(*
Nazwa:		FB_WeightStation
Opis:		Podnoszenie wag
Wersja:		V0.26
Data:		04.09.2024
Autor:		DP, 
Urządzenia:	Siłowniki
Ostatnie zmiany:
	- 20250904 [DP] EventLog-do sprawdzenia, 1 spr->wywołać błędy 
	- 2024-10-01 [DP] Liczniki po Aborting
	- 2024-04-17 [DP] Przerobienie liczenia i uprowszenie, dwufaz

Konfiguracja:
	- Krokówka
	Instukcja:
		-
		-
	
Info:
	- 
*)

FUNCTION_BLOCK FB_WeightStation
VAR_INPUT
	bEnable											: BOOL;
	bEStop											: BOOL;
	bRun											: BOOL;

	bTwoPhaseMode									: BOOL;
	bCountingBeforeSensorsMode						: BOOL;
    eGlobalState        							: E_PMLState; 							//Stan ogólny maszyny, tylko do błędu
	bConveyorRunning								: BOOL;									//Transporter pracuje, tylko do błędu
	bWeight1ActuatorSensorUp						: BOOL;									//Pierwsza waga podniesiona
	bWeight1FormSensor								: BOOL;									//Obecność formatki na pierwszej wadze     
	bWeight1FormBeforeSensor						: BOOL;									//Obecność formatki przed pierwszą wagą 

	bWeight2ActuatorSensorUp						: BOOL;									//Druga waga podniesiona
	bWeight2FormSensor								: BOOL;									//Obecność formatki na drugiek wadze
	bWeight2FormBeforeSensor						: BOOL;									//Obecność formatki przed pierwszą wagą 
	
	bWeight3ActuatorSensorUp						: BOOL;									//Trzecia waga podniesiona
	bWeight3FormSensor								: BOOL;									//Obecność formatki na trzeciej wadze
	bWeight3FormBeforeSensor						: BOOL;									//Obecność formatki przed pierwszą wagą 
	
	bWeight4ActuatorSensorUp						: BOOL;									//Czwarta waga podniesiona
	bWeight4FormSensor								: BOOL;									//Obecność formatki na czwartej wadze
	bWeight4FormBeforeSensor						: BOOL;									//Obecność formatki przed pierwszą wagą 
	
	bCanReleaseForms								: BOOL;									//Można wypuścić formatki
	bWeighingCycle									: BOOL;									//Trwa ważenie
                                    	
	arrWeightPackageState							: ARRAY [1..17] OF S_PackageState;		//Rejestr nad wagami
	
	bResetCycle										: BOOL;									//Reset cyklu
	
	bHoming											: BOOL;
	bIgnoreError									: BOOL;
	bReset											: BOOL;
	bManualMovement									: BOOL;
	                                    			
	_TIMERS_										: BOOL;
	tWeight1ActuatorUpDelay							: TIME;									//Opóźnienie podnoszenia wagi 1
	tWeight2ActuatorUpDelay							: TIME;									//Opóźnienie podnoszenia wagi 2
	tWeight3ActuatorUpDelay							: TIME;									//Opóźnienie podnoszenia wagi 3
	tWeight4ActuatorUpDelay							: TIME;									//Opóźnienie podnoszenia wagi 4
	
	_ALARMINFO_										: BOOL;
	udiStationIndex									: UDINT;								//Numer stacji
	sStationName									: WSTRING;
	
END_VAR   
                              			
VAR_OUTPUT                              			
	eState											: E_Station;							//Stan ogólny bloku
	eRunningState									: E_WeightLiftStationState;				//Stan stacji
	
	bWeight1Actuator								: BOOL;									//Podnoszenie 1 wagi
	bWeight2Actuator								: BOOL;									//Podnoszenie 2 wagi
	bWeight3Actuator								: BOOL;									//Podnoszenie 3 wagi
	bWeight4Actuator								: BOOL;									//Podnoszenie 4 wagi

	iFormsCounterWeight1							: INT;									//Licznik formatek
	iFormsCounterWeight2							: INT;									//Licznik formatek na wadze 2
	iFormsCounterWeight3							: INT;									//Licznik formatek na wadze 3
	iFormsCounterWeight4							: INT;									//Licznik formatek na wadze 4
	
	bError											: BOOL;									//Błąd stacji
	udiErrorID										: UDINT;								//Numer błędu
	sErrorDescription								: STRING(255);							//Opis błędu
	sErrorDescription2								: STRING(200);							//Opis błędu
	sErrorStationName								: STRING(200);							//Nazwa stacji
	udiStationID									: UDINT;								// Nr stacji
                                    			
	tCycleTime										: TIME;									//Czas cyklu
	bHomingDone										: BOOL;									//Stacja zbazowana 
	bWeighingCycleDone								: BOOL;									//Koniec ważenia 
	bCycleDone										: BOOL;									//Cykl skończony 			
	bTareWeights									: BOOL;		
END_VAR

VAR_IN_OUT
	bManualWeight1Actuator							: BOOL;									//Tryb manualny, Waga 1 UP	
	bManualWeight2Actuator							: BOOL;									//Tryb manualny, Waga 2 UP
	bManualWeight3Actuator							: BOOL;									//Tryb manualny, Waga 3 UP
	bManualWeight4Actuator							: BOOL;									//Tryb manualny, Waga 4 UP	
	bDeparture										: BOOL;					
	bAutoTare										: BOOL;	
END_VAR

VAR
	eLastStateTemp									: E_Station;							//Ostatni stan CONTROL
	eLastState										: E_Station;							//Ostatni stan CONTROL
	eLastRunningStateTemp							: E_WeightLiftStationState;				//Ostatni stan Running
	eLastRunningState								: E_WeightLiftStationState;				//Ostatni stan Running
	eRunningStateBeforeEStop	             		: E_WeightLiftStationState;	                      			                                    		
	tonWeight1ActuatorDelay							: TON;									//TON, opóźnienie podnoszenia wagi 1
	tonWeight2ActuatorDelay							: TON;									//TON, opóźnienie podnoszenia wagi 2
	tonWeight3ActuatorDelay							: TON;									//TON, opóźnienie podnoszenia wagi 3
	tonWeight4ActuatorDelay							: TON;									//TON, opóźnienie podnoszenia wagi 4
	tonWeightAntuatorOffDelay						: TON;
	tonPreparingToReadyDelay						: TON;
	tonResetting									: TON;
	tofRunning										: TOF;
	rtResetCommands									: R_TRIG;
	tonHoming 										: TON;
	tonReadyAndRepair								: TON;					
	tonAbortedDelay									: TON;
	tonRepairDelay									: TON;									//TON, czas po którym przechodzimy do naprawy
	tonRepairOnDelay								: TON;									//TON, czas na wyjazd wszystkich formatek
	rtWeight1FormSensor								: R_TRIG;								//R_Trig, zbocze nar (przy wadze 1)
	rtWeight2FormSensor								: R_TRIG;								//R_Trig, zbocze nar (przy wadze 2)
	rtWeight3FormSensor								: R_TRIG;								//R_Trig, zbocze nar (przy wadze 3)
	rtWeight4FormSensor								: R_TRIG;								//R_Trig, zbocze nar (przy wadze 4)

	ftWeight1FormBeforeSensor						: F_TRIG;								
	ftWeight2FormBeforeSensor						: F_TRIG;								
	ftWeight3FormBeforeSensor						: F_TRIG;								
	ftWeight4FormBeforeSensor						: F_TRIG;								
	
	tonWeightsEmpty									: TON;
	toniCaseTareWeights1							: TON;
	toniCaseTareWeights2							: TON;
	
	bLastStateWeight1Actuator						: BOOL;							
	bLastStateWeight2Actuator						: BOOL;	
	bLastStateWeight3Actuator						: BOOL;	
	bLastStateWeight4Actuator						: BOOL;	
	
	bStateError										: BOOL;
	bWasAborting									: BOOL;
	
	bRepairAllRegistersAreEmpty						: BOOL;								
	
	//Błedy
	bResetCycleOn									: BOOL;
	tonWeight1ActuatorUpError 						: TON;
	tonWeight2ActuatorUpError 						: TON;
	tonWeight3ActuatorUpError 						: TON;
	tonWeight4ActuatorUpError 						: TON;
	
	//Śmiecie
	tonRepair1: TON;
	tonRepair2: TON;
	tonRepair3: TON;
	tonRepair4: TON;
	tonRepair5: TON;
	tonRepair6: TON;
	
	rtrigCycleTimerRead: R_TRIG;
	tonCycleTimer: TON;
	tt: INT;
	rtWeight3FormSensorWithDelay2: R_TRIG;

	iRepair1: INT;
	iRepair2: INT;
	iRepair3: INT;
	iRepair4: INT;
	iRepair5: INT;
	iRepair6: INT;
	
	tofRunningStopping: TOF;
	iCaseTareWeights:INT;
	
	//Zmienne od EVENTLOGGER
	bAlarmInit 						: BOOL := TRUE; 
	nAlarmNumerator					: INT;
	arfbAlarm						: ARRAY[0..19] OF  FB_TcAlarm;		//Tablica bloczków błędów
	fbSourceInfo 					: FB_TcSourceInfo;
	iSourceInfo						: I_TcSourceInfo;
	sAlarmTest						: STRING;
	tonEventLogger					: TON;
	//Koniec zmiennych od EVENTLOGGER
	bTest							: BOOL;
END_VAR

ResetAll();
ACT_ErrorHandling();
ACT_Signals();
aRepair();
ACT_Control();
ACT_Statistics();
aStationID();

IF eLastStateTemp <> eState THEN
	eLastState							:= eLastStateTemp;
END_IF
eLastStateTemp							:= eState;

IF eLastRunningStateTemp <> eRunningState THEN
	eLastRunningState					:= eLastRunningStateTemp;
END_IF
eLastRunningStateTemp					:= eRunningState;

ACTION ACT_Control:


	(*****Wyłączenie enable*****)
	IF NOT bEnable AND NOT bError THEN
		IF eState <> E_Station.eDisabled AND eState <> E_Station.ePreparingToDisable THEN
				eState 								:= E_Station.ePreparingToDisable; 
		END_IF	
	END_IF

	(*****Estop*****)
	IF NOT bEstop  THEN	
		IF eState <> E_Station.eAborted AND eState <> E_Station.eAborting AND eState <> E_Station.eDisabled THEN
				eRunningStateBeforeEStop			:= eRunningState;
				eState 								:= E_Station.eAborting; 
		END_IF
	END_IF


CASE eState OF
	
	
	E_Station.eDisabled: 					// Stan nieaktywnosci (Stacja wyłączona)
		IF bEnable THEN
			eState											:= E_Station.ePreparingToReady;
		END_IF	
	//------------------------------------------------------------------------------
	
	E_Station.eAborted: 					// Stan bezpiecznego zatrzymania (po Abortingu)			
		IF bEStop THEN
			eState											:= E_Station.ePreparingToReady;
		END_IF	
	//------------------------------------------------------------------------------
	
	E_Station.eAborting:                 	// Stan bezpiecznego zatrzymywania (po EStopie)
	
		aResetCommandsAborting();
		bWasAborting										:= TRUE;
		eState												:= E_Station.eAborted;	
		eRunningState										:= E_WeightLiftStationState.eReady;
	//------------------------------------------------------------------------------
	
	E_Station.eError:                 	 	// Stan błędu 	
	
		IF bReset THEN
			eState									:= E_Station.eResetting;	
		ELSE
			aResetCommands();
		END_IF
		
	//------------------------------------------------------------------------------

	
	E_Station.eResetting:					// Stan resetowania bledu (po Errorze)

// 		CASE udiErrorID OF 
// //		CASE udiErrorID - udiStationIndex OF 
// 			
// 			191,195: //Error 1
// 				bWeight1Actuator						:=	FALSE;
// 				bError									:=	FALSE;
// 			192,196://Error 2
// 				bWeight2Actuator						:=	FALSE;
// 				bError									:=	FALSE;	
// 			193: //Error 3
// 				bWeight3Actuator						:=	FALSE;
// 				bError									:=	FALSE;
// 			194: //Error 4
// 				bWeight4Actuator						:=	FALSE;
// 				bError									:=	FALSE;			
// 			
// 		END_CASE

		bWeight1Actuator						:=	FALSE;
		bWeight2Actuator						:=	FALSE;		
		bWeight3Actuator						:=	FALSE;
		bWeight4Actuator						:=	FALSE;		

		IF NOT bError THEN
			udiErrorID										:= 0;
			sErrorDescription								:= '';
			sErrorDescription2								:= '';
			eState											:= E_Station.ePreparingToReady;
		ELSIF tonResetting.Q THEN                   	
			eState											:= E_Station.eError;
		END_IF
	//------------------------------------------------------------------------------
	E_Station.eManualMovement:     			// Stan ruchów manualnych  
	
		ACT_ManualMovements();
		//Wyjście z trybu serwisowego
		IF NOT bManualMovement THEN
			bWeight1Actuator								:=	bLastStateWeight1Actuator;
			bWeight2Actuator								:=	bLastStateWeight2Actuator;
			bWeight3Actuator								:=	bLastStateWeight3Actuator;
			bWeight4Actuator								:=	bLastStateWeight4Actuator;
			eState											:=	E_Station.eReady;
		END_IF
	//------------------------------------------------------------------------------
	
	E_Station.eHoming:						// Stan bazowania
	
		ACT_Homing();
		IF NOT bHoming AND tonHoming.Q THEN
			eState									:=	E_Station.ePreparingToReady;
		END_IF	
	//------------------------------------------------------------------------------
	
	E_Station.eHomingDone:                  // Stan wykonania bazowania
	
		bHomingDone											:= TRUE;		
		IF NOT bHoming THEN
			eState											:= E_Station.eReady;
		END_IF	
	//------------------------------------------------------------------------------
	
	
	E_Station.ePreparingToReady:            // Stan przygotowywania do gotowosci (zawsze przed Ready)
		//bHomingDone										:=	FALSE;	
		bWeight1Actuator									:=	FALSE;
		bWeight2Actuator									:=	FALSE;
		bWeight3Actuator									:=	FALSE;
		bWeight4Actuator									:=	FALSE;
		
		IF NOT bWasAborting THEN
			iFormsCounterWeight1								:= 3;	
			iFormsCounterWeight2								:= 2;
			iFormsCounterWeight3								:= 1;
			iFormsCounterWeight4								:= 0;
		END_IF
		
		IF tonPreparingToReadyDelay.Q THEN
			eState											:= E_Station.eReady;
		END_IF	
		
	//------------------------------------------------------------------------------
	
	
	E_Station.ePreparingToDisable:          // Stan przygotowywania do nieaktywnosci (po wyłączeniu Enable)	
		
		bWeight1Actuator									:=	FALSE;
		bWeight2Actuator									:=	FALSE;
		bWeight3Actuator									:=	FALSE;
		bWeight4Actuator									:=	FALSE;
		
		iFormsCounterWeight1								:= 3;	
		iFormsCounterWeight2								:= 2;
		iFormsCounterWeight3								:= 1;
		iFormsCounterWeight4								:= 0;
					
		eState												:= E_Station.eDisabled;
		eRunningState										:= E_WeightLiftStationState.eDisabled;
		
	//------------------------------------------------------------------------------
	
	
	E_Station.eReady:						// Stan gotowosci
		bWasAborting										:= FALSE;
		IF (bRun OR bAutoTare) AND bHomingDone AND NOT bCycleDone THEN
			eRunningState									:= E_WeightLiftStationState.eReady;
			eState											:= E_Station.eStarting;
		END_IF
		
		IF bHoming THEN
			eState											:= E_Station.eHoming;
		END_IF
		
		IF bManualMovement THEN
			bLastStateWeight1Actuator	:=	bManualWeight1Actuator	:=	bWeight1Actuator;
			bLastStateWeight2Actuator	:=	bManualWeight2Actuator	:=	bWeight2Actuator;
			bLastStateWeight3Actuator	:=	bManualWeight3Actuator	:=	bWeight3Actuator;
			bLastStateWeight4Actuator	:=	bManualWeight4Actuator	:=	bWeight4Actuator;		
			eState											:= E_Station.eManualMovement;
		END_IF
		
		IF NOT bRun THEN
			bCycleDone										:= FALSE;
		END_IF
		IF tonReadyAndRepair.Q THEN
			eRunningState									:= E_WeightLiftStationState.eReady;
		END_IF
	//------------------------------------------------------------------------------
	
	
	E_Station.eStopping:					// Stan zatrzymywania 

		ACT_Running();
		eState											:= E_Station.eReady;
		eRunningState									:= E_WeightLiftStationState.eReady;
		
		
	//------------------------------------------------------------------------------
	
	
	E_Station.eStarting:                  	// Stan uruchamiania (po Ready)
	
		eState												:= E_Station.eRunning;
	//------------------------------------------------------------------------------
	
	
	E_Station.eRunning:               		// Stan wykonywania cyklu (po Startingu), w tym stanie osobny
		
		ACT_Running();
		
		IF NOT bRun THEN
			eState											:= E_Station.eStopping;
		END_IF
		
		IF bCycleDone THEN
			eState											:= E_Station.eReady;
		END_IF
	//------------------------------------------------------------------------------
	
	
END_CASE
END_ACTION

ACTION ACT_ErrorHandling:
// Alarm_0300	300	Error	Podnoszenie wagi nr 1 | Blokada podnoszenia siłownika - sprawdź czujnik lub odblokuj
// Alarm_0301	301	Error	Podnoszenie wagi nr 2 | Blokada podnoszenia siłownika - sprawdź czujnik lub odblokuj
// Alarm_0302	302	Error	Podnoszenie wagi nr 3 | Blokada podnoszenia siłownika - sprawdź czujnik lub odblokuj
// Alarm_0303	303	Error	Podnoszenie wagi nr 4 | Blokada podnoszenia siłownika - sprawdź czujnik lub odblokuj
// Alarm_0304	304	Error	Podnoszenie wagi nr 5 | Blokada podnoszenia siłownika - sprawdź czujnik lub odblokuj
// Alarm_0305	305	Error	Podnoszenie wagi nr 6 | Blokada podnoszenia siłownika - sprawdź czujnik lub odblokuj

IF bAlarmInit THEN
    bAlarmInit := FALSE; 
	fbSourceInfo.Clear();
	fbSourceInfo.sName:=wsLiteral_TO_UTF8(sStationName);//'Machine';
	fbSourceInfo.nId:=udiStationIndex;//2700;
	// Alarm_0300	300	Error	Podnoszenie wagi nr 1 | Blokada podnoszenia siłownika - sprawdź czujnik lub odblokuj
    arfbAlarm[0].CreateEx(stEventEntry := TC_EVENTS.AlarmClass.Alarm_0300, bWithConfirmation:= FALSE,  ipSourceInfo:= fbSourceInfo); 
	// Alarm_0301	301	Error	Podnoszenie wagi nr 2 | Blokada podnoszenia siłownika - sprawdź czujnik lub odblokuj
	arfbAlarm[1].CreateEx(stEventEntry := TC_EVENTS.AlarmClass.Alarm_0301, bWithConfirmation:= FALSE,  ipSourceInfo:= fbSourceInfo);
	// Alarm_0302	302	Error	Podnoszenie wagi nr 3 | Blokada podnoszenia siłownika - sprawdź czujnik lub odblokuj
	arfbAlarm[2].CreateEx(stEventEntry := TC_EVENTS.AlarmClass.Alarm_0302, bWithConfirmation:= FALSE,  ipSourceInfo:= fbSourceInfo);
	// Alarm_0303	303	Error	Podnoszenie wagi nr 4 | Blokada podnoszenia siłownika - sprawdź czujnik lub odblokuj
	arfbAlarm[3].CreateEx(stEventEntry := TC_EVENTS.AlarmClass.Alarm_0303, bWithConfirmation:= FALSE,  ipSourceInfo:= fbSourceInfo);
	// Alarm_0304	304	Error	Podnoszenie wagi nr 5 | Blokada podnoszenia siłownika - sprawdź czujnik lub odblokuj
	arfbAlarm[4].CreateEx(stEventEntry := TC_EVENTS.AlarmClass.Alarm_0304, bWithConfirmation:= FALSE,  ipSourceInfo:= fbSourceInfo);
	// Alarm_0305	305	Error	Podnoszenie wagi nr 6 | Blokada podnoszenia siłownika - sprawdź czujnik lub odblokuj
	arfbAlarm[5].CreateEx(stEventEntry := TC_EVENTS.AlarmClass.Alarm_0305, bWithConfirmation:= FALSE,  ipSourceInfo:= fbSourceInfo);
END_IF

bStateError								:= (eState = E_Station.eError) OR (eState = E_Station.eResetting);

tonEventLogger (IN:= NOT tonEventLogger.Q, PT:=T#1S);

IF tonEventLogger.Q THEN
	
	// Alarm_0300	300	Error	Podnoszenie wagi nr 1 | Blokada podnoszenia siłownika - sprawdź czujnik lub odblokuj
	// Alarm_0304	304	Error	Podnoszenie wagi nr 5 | Blokada podnoszenia siłownika - sprawdź czujnik lub odblokuj
	//Błąd podnoszenia wagi 1 
	tonWeight1ActuatorUpError				(IN:= bWeight1Actuator AND NOT bWeight1ActuatorSensorUp	, PT:=T#2S);
	IF tonWeight1ActuatorUpError.Q THEN
		IF NOT bTwoPhaseMode AND NOT arfbAlarm[0].bActive THEN
			arfbAlarm[0].Raise(nTimeStamp:=0);
		END_IF
		IF bTwoPhaseMode AND NOT arfbAlarm[4].bActive THEN
				arfbAlarm[4].Raise(nTimeStamp:=0);
		END_IF
		IF (arfbAlarm[0].bActive OR arfbAlarm[4].bActive) AND bReset THEN
			bWeight1Actuator			:= FALSE;
		END_IF
		ELSE	
		IF NOT bTwoPhaseMode AND arfbAlarm[0].bActive AND bReset THEN
			arfbAlarm[0].Clear(nTimeStamp:=0, bResetConfirmation:= FALSE);
		END_IF
		IF bTwoPhaseMode AND arfbAlarm[4].bActive AND bReset THEN
			arfbAlarm[4].Clear(nTimeStamp:=0, bResetConfirmation:= FALSE);
		END_IF
	// 	bError								:= TRUE;
	// 	IF NOT bTwoPhaseMode THEN
	// 	udiErrorID							:= 191;	
	// 	//udiErrorID 						:= udiErrorID + udiStationIndex;
	// 	sErrorDescription					:= 'Podnoszenie wagi nr 1';
	// 	END_IF
	// 	
	// 	IF bTwoPhaseMode THEN
	// 		udiErrorID						:= 195;
	// 		sErrorDescription				:= 'Podnoszenie wagi nr 5';
	// 	END_IF
	// 	sErrorDescription2					:= 'Blokada podnoszenia siłownika - sprawdź czujnik lub odblokuj';
	END_IF
	// Alarm_0301	301	Error	Podnoszenie wagi nr 2 | Blokada podnoszenia siłownika - sprawdź czujnik lub odblokuj
	// Alarm_0305	305	Error	Podnoszenie wagi nr 6 | Blokada podnoszenia siłownika - sprawdź czujnik lub odblokuj
	//Błąd podnoszenia wagi 2
	tonWeight2ActuatorUpError				(IN:= bWeight2Actuator AND NOT bWeight2ActuatorSensorUp	, PT:=T#2S);
	IF tonWeight2ActuatorUpError.Q THEN
		
		IF NOT bTwoPhaseMode AND NOT arfbAlarm[1].bActive THEN
				arfbAlarm[1].Raise(nTimeStamp:=0);
		END_IF
		IF bTwoPhaseMode AND NOT arfbAlarm[5].bActive THEN
				arfbAlarm[5].Raise(nTimeStamp:=0);
		END_IF	
		IF (arfbAlarm[1].bActive OR arfbAlarm[5].bActive) AND bReset THEN
			bWeight1Actuator			:= FALSE;
		END_IF
		ELSE	
		IF NOT bTwoPhaseMode AND arfbAlarm[1].bActive AND bReset THEN
			arfbAlarm[1].Clear(nTimeStamp:=0, bResetConfirmation:= FALSE);
		END_IF	
		IF bTwoPhaseMode AND arfbAlarm[5].bActive AND bReset THEN
			arfbAlarm[5].Clear(nTimeStamp:=0, bResetConfirmation:= FALSE);
		END_IF	
	// 	bError								:= TRUE;
	// 	IF NOT bTwoPhaseMode THEN
	// 	udiErrorID							:= 192;	
	// 	//udiErrorID 						:= udiErrorID + udiStationIndex;
	// 	sErrorDescription					:= 'Podnoszenie wagi nr 2';
	// 	END_IF
	
	// 	IF bTwoPhaseMode THEN
	// 		udiErrorID						:= 196;
	// 		sErrorDescription				:= 'Podnoszenie wagi nr 6';
	// 	END_IF
	// 	sErrorDescription2					:= 'Blokada podnoszenia siłownika - sprawdź czujnik lub odblokuj';	
	END_IF
	// Alarm_0302	302	Error	Podnoszenie wagi nr 3 | Blokada podnoszenia siłownika - sprawdź czujnik lub odblokuj
	//Błąd podnoszenia wagi 3
	tonWeight3ActuatorUpError				(IN:= bWeight3Actuator AND NOT bWeight3ActuatorSensorUp	OR bTest, PT:=T#2S);
	IF tonWeight3ActuatorUpError.Q THEN
		IF NOT arfbAlarm[2].bActive THEN
				arfbAlarm[2].Raise(nTimeStamp:=0);
			END_IF
		ELSE	
			IF  arfbAlarm[2].bActive AND bReset THEN
				arfbAlarm[2].Clear(nTimeStamp:=0, bResetConfirmation:= FALSE);
			END_IF	
	// 	bError								:= TRUE;
	// 	udiErrorID							:= 193;	
	// 	//udiErrorID 						:= udiErrorID + udiStationIndex;
	// 	sErrorDescription					:= 'Podnoszenie wagi nr 3';
	// 	sErrorDescription2					:= 'Blokada podnoszenia siłownika - sprawdź czujnik lub odblokuj';
	END_IF
	// Alarm_0303	303	Error	Podnoszenie wagi nr 4 | Blokada podnoszenia siłownika - sprawdź czujnik lub odblokuj
	//Błąd podnoszenia wagi 4
	tonWeight4ActuatorUpError				(IN:= bWeight4Actuator AND NOT bWeight4ActuatorSensorUp	, PT:=T#2S);
	IF tonWeight4ActuatorUpError.Q THEN
		IF NOT arfbAlarm[3].bActive THEN
				arfbAlarm[3].Raise(nTimeStamp:=0);
			END_IF
		ELSE	
			IF  arfbAlarm[3].bActive AND bReset THEN
				arfbAlarm[3].Clear(nTimeStamp:=0, bResetConfirmation:= FALSE);
			END_IF	
	// 	bError								:= TRUE;
	// 	udiErrorID							:= 194;	
	// 	//udiErrorID 						:= udiErrorID + udiStationIndex;
	// 	sErrorDescription					:= 'Podnoszenie wagi nr 4';
	// 	sErrorDescription2					:= 'Blokada podnoszenia siłownika - sprawdź czujnik lub odblokuj';
	END_IF
	
	IF NOT bEnable OR NOT bEStop THEN
		bError								:= FALSE;
	END_IF
	
	IF bError AND NOT bStateError THEN
		eState								:= E_Station.eError;
	END_IF
	
	(*Przepisywanie nazwy stacji*)
	sErrorStationName						:= WSTRING_TO_STRING(sStationName);
	
	(*Wyświetlanie błedu na wyjściu*)
	bError									:= FALSE;
	
	FOR nAlarmNumerator := 0 TO 19 DO
		bError								:= bError OR arfbAlarm[nAlarmNumerator].bActive;
	END_FOR
END_IF
END_ACTION

ACTION ACT_Homing:
bWeight1Actuator						:= FALSE;
bWeight2Actuator						:= FALSE;
bWeight3Actuator						:= FALSE;
bWeight4Actuator						:= FALSE;

iFormsCounterWeight1					:= 0;
iFormsCounterWeight2					:= 1;
iFormsCounterWeight3					:= 2;
iFormsCounterWeight4					:= 3;

eState									:= E_Station.eHomingDone;
END_ACTION

ACTION ACT_ManualMovements:


IF NOT bRun (*AND bManualMovement*) THEN
	
	bWeight1Actuator		:=	bManualWeight1Actuator;
	bWeight2Actuator		:=	bManualWeight2Actuator;
	bWeight3Actuator		:=	bManualWeight3Actuator;
	bWeight4Actuator		:=	bManualWeight4Actuator;	
ELSE
	bManualWeight1Actuator	:=	FALSE;
	bManualWeight2Actuator	:=	FALSE;
	bManualWeight3Actuator	:=	FALSE;
	bManualWeight4Actuator	:=	FALSE;		
END_IF


IF bHoming THEN
	eState											:= E_Station.eHoming;
END_IF

//Running();

IF NOT bRun THEN
	bCycleDone 										:= FALSE;
END_IF
END_ACTION

ACTION ACT_Running:

CASE eRunningState OF
	
	E_WeightLiftStationState.eRepair:		//Naprawa
		
		bWeight1Actuator								:= FALSE;
		bWeight2Actuator								:= FALSE;
		bWeight3Actuator								:= FALSE;
		bWeight4Actuator								:= FALSE;
		
		iFormsCounterWeight4							:= 0;	
		iFormsCounterWeight3							:= 1;
		iFormsCounterWeight2							:= 2;
		iFormsCounterWeight1							:= 3;
		
		IF bTwoPhaseMode THEN
			iFormsCounterWeight2						:= 0;
			iFormsCounterWeight1						:= 1;
		END_IF
		
		IF NOT arrWeightPackageState[1].bFormPresent AND NOT arrWeightPackageState[2].bFormPresent AND NOT arrWeightPackageState[3].bFormPresent AND NOT arrWeightPackageState[4].bFormPresent THEN
			
			IF tonRepairOnDelay.Q THEN
				eRunningState							:= E_WeightLiftStationState.ePrepareToStorageOfForms;	
			END_IF
	
		END_IF
		

	E_WeightLiftStationState.eDisabled :	//Stan wyłączony
	
		eRunningState									:= E_WeightLiftStationState.eReady;
		
	//----------------------------------------------------------------------------------------
		
	E_WeightLiftStationState.eReady :		//Sprawdzam co się dzieje ze stacją
	
(*	w1
		//IF bDeparture THEN
			
			//eRunningState								:= E_WeightLiftStationState.ePrepareToStorageOfForms;
			
		IF NOT bWeight1FormSensor AND NOT bWeight2FormSensor AND NOT bWeight3FormSensor AND NOT bWeight4FormSensor THEN //Nie ma wszystkich formatek
		
			iFormsCounterWeight4						:= 0;	
			iFormsCounterWeight3						:= 1;
			iFormsCounterWeight2						:= 2;
			iFormsCounterWeight1						:= 3;
			eRunningState								:= E_WeightLiftStationState.ePrepareToStorageOfForms;

		//Przechodzę do opuszczanie formatek
		ELSIF bWeight1FormSensor AND bWeight2FormSensor AND bWeight3FormSensor AND bWeight4FormSensor THEN //Mamy wszystkie formateki
			
			iFormsCounterWeight4						:= 0;	
			iFormsCounterWeight3						:= 0;
			iFormsCounterWeight2						:= 0;
			iFormsCounterWeight1						:= 0;
			eRunningState								:= E_WeightLiftStationState.eWeighingCycleON;	
			
		ELSE
			//eRunningState								:= E_WeightLiftStationState.eRepair;
			eRunningState								:= E_WeightLiftStationState.ePrepareToStorageOfForms;			
		END_IF
*)		

	(*	w2	*)
		
		IF NOT bAutoTare THEN
			eRunningState								:= E_WeightLiftStationState.ePrepareToStorageOfForms;		
		ELSE
			CASE iCaseTareWeights OF
				0:
					iCaseTareWeights	:=	iCaseTareWeights	+	10;
				10:
				 IF tonWeightsEmpty.Q THEN
					 iCaseTareWeights	:=	iCaseTareWeights	+	10;
				 END_IF
				20:
					bWeight1Actuator	:= TRUE;
					bWeight2Actuator	:= TRUE;
					bWeight3Actuator	:= NOT bTwoPhaseMode;
					bWeight4Actuator	:= NOT bTwoPhaseMode;				
					iCaseTareWeights	:= iCaseTareWeights	+	10;
				30:
					IF toniCaseTareWeights1.Q THEN
						iCaseTareWeights:=	iCaseTareWeights	+	10;
					END_IF
				40:
					bTareWeights		:= TRUE;
					iCaseTareWeights	:= iCaseTareWeights	+	10;	
				50:
					IF toniCaseTareWeights2.Q THEN
						bAutoTare		:= FALSE;
						bTareWeights	:= FALSE;
						iCaseTareWeights:= 0;
					END_IF				
			END_CASE
		END_IF
		
		
		
	//----------------------------------------------------------------------------------------	

	E_WeightLiftStationState.ePrepareToStorageOfForms: //Przygotowywanie do magazynowania formatek
		
		bWeight1Actuator								:= FALSE;
		bWeight2Actuator								:= FALSE;
		bWeight3Actuator								:= FALSE;
		bWeight4Actuator								:= FALSE;
		
		eRunningState									:=  E_WeightLiftStationState.eStorageOfForms;	
	//----------------------------------------------------------------------------------------		
	
	E_WeightLiftStationState.eStorageOfForms:	//Magazynuje formatki
		
		//Waga 1/5====================================================================================================================
		IF (tonWeight1ActuatorDelay.Q OR bCountingBeforeSensorsMode) AND ((	iFormsCounterWeight1 = 4 AND NOT	bTwoPhaseMode) OR 
																			iFormsCounterWeight1 = 2 AND 		bTwoPhaseMode) THEN	
			bWeight1Actuator	:= TRUE;
		END_IF
		
		//Waga 2/6=====================================================================================================================		
		IF (tonWeight2ActuatorDelay.Q OR bCountingBeforeSensorsMode) AND ((	iFormsCounterWeight2 = 4  AND NOT	bTwoPhaseMode) OR 
																			iFormsCounterWeight2 = 2 AND 		bTwoPhaseMode) THEN	
			bWeight2Actuator	:= TRUE;
		END_IF
		
		//Waga 3====================================================================================================================
		IF (tonWeight3ActuatorDelay.Q OR bCountingBeforeSensorsMode) AND iFormsCounterWeight3 = 4	THEN //Podnoszenie Waga 3
			bWeight3Actuator	:= NOT bTwoPhaseMode;
		END_IF
			
		//Waga 4=====================================================================================================================	
		IF (tonWeight4ActuatorDelay.Q OR bCountingBeforeSensorsMode) AND iFormsCounterWeight4 = 4	THEN //Podnoszenie Waga 4
			bWeight4Actuator	:= NOT bTwoPhaseMode;
		END_IF

		
		IF (bWeight1ActuatorSensorUp) AND (bWeight2ActuatorSensorUp) AND
 		   (bWeight3ActuatorSensorUp OR bTwoPhaseMode) AND (bWeight4ActuatorSensorUp OR bTwoPhaseMode) THEN
		   		eRunningState								:= E_WeightLiftStationState.eWeighingCycleStart;
		   
		END_IF
		
	//----------------------------------------------------------------------------------------
	
	E_WeightLiftStationState.eWeighingCycleStart:	//Rozpoczęcie Ważenia
	
		IF bWeighingCycle THEN
			eRunningState								:= E_WeightLiftStationState.eWeighingCycleON;
		END_IF

	//----------------------------------------------------------------------------------------

	
	E_WeightLiftStationState.eWeighingCycleON:	//Trwa ważenie
	
		IF (arrWeightPackageState[1].bWeighed OR arrWeightPackageState[1].bWeightAborted) AND (arrWeightPackageState[2].bWeighed OR arrWeightPackageState[2].bWeightAborted) AND
		   (arrWeightPackageState[3].bWeighed OR arrWeightPackageState[3].bWeightAborted OR bTwoPhaseMode) AND (arrWeightPackageState[4].bWeighed OR arrWeightPackageState[4].bWeightAborted OR bTwoPhaseMode) THEN  //Czekam na przepisanie statusów z wag
		   bWeighingCycleDone	:=	TRUE;
			IF bCanReleaseForms THEN			//Mogę wypuścić formatki
				eRunningState							:= E_WeightLiftStationState.eWeightLiftDown;
				bWeighingCycleDone	:=	FALSE;
			END_IF
			
		END_IF
	//----------------------------------------------------------------------------------------
	
	
	E_WeightLiftStationState.eWeightLiftDown:	//Opuszczanie formatek
		
		bWeight1Actuator								:= FALSE;
		bWeight2Actuator								:= FALSE;
		bWeight3Actuator								:= FALSE;
		bWeight4Actuator								:= FALSE;
		
		iFormsCounterWeight4							:= 0;	
		iFormsCounterWeight3							:= 0;
		iFormsCounterWeight2							:= 0;
		iFormsCounterWeight1							:= 0;
		
		IF tonWeightAntuatorOffDelay.Q THEN	        
			eRunningState								:= E_WeightLiftStationState.eDepartureOfForms;
		END_IF	
	//----------------------------------------------------------------------------------------
	
	E_WeightLiftStationState.eDepartureOfForms:	//Wypuszczamy formatki

			eRunningState								:= E_WeightLiftStationState.eDone;
			bDeparture									:= TRUE;

	//----------------------------------------------------------------------------------------
	
	E_WeightLiftStationState.eDone:				//Cykl skończony
		
			bCycleDone									:= TRUE;		//Wystawiam koniec cyklu
			eRunningState								:= E_WeightLiftStationState.eReady;
		
			
END_CASE
END_ACTION

ACTION ACT_Signals:
//TONs
tonWeight1ActuatorDelay		(IN:= eRunningState = E_WeightLiftStationState.eStorageOfForms AND bWeight1FormSensor, PT:= tWeight1ActuatorUpDelay);
tonWeight2ActuatorDelay		(IN:= eRunningState = E_WeightLiftStationState.eStorageOfForms AND bWeight2FormSensor, PT:= tWeight2ActuatorUpDelay);
tonWeight3ActuatorDelay		(IN:= eRunningState = E_WeightLiftStationState.eStorageOfForms AND bWeight3FormSensor, PT:= tWeight3ActuatorUpDelay);
tonWeight4ActuatorDelay		(IN:= eRunningState = E_WeightLiftStationState.eStorageOfForms AND bWeight4FormSensor, PT:= tWeight4ActuatorUpDelay);
tonWeightAntuatorOffDelay 	(IN:= NOT bWeight1Actuator AND NOT bWeight2Actuator AND NOT bWeight3Actuator AND NOT bWeight4Actuator, PT:=T#100MS);

tonPreparingToReadyDelay	(IN:= eState = E_Station.ePreparingToReady			,PT:= T#300MS);
tonResetting				(IN:= eState = E_Station.eResetting					,PT:= T#200MS);
tonHoming					(IN:= eState = E_Station.eHoming					,PT:= T#1S);
rtResetCommands				(CLK:=eState = E_Station.eReady 					,Q=>); 
tonReadyAndRepair			(IN:= eState = E_Station.eReady AND eRunningState = E_WeightLiftStationState.eRepair, PT:=T#10S);
//Triggers

rtWeight1FormSensor			(CLK:= bWeight1FormSensor AND NOT bCountingBeforeSensorsMode);
rtWeight2FormSensor			(CLK:= bWeight2FormSensor AND NOT bCountingBeforeSensorsMode);
rtWeight3FormSensor			(CLK:= bWeight3FormSensor AND NOT bCountingBeforeSensorsMode);
rtWeight4FormSensor			(CLK:= bWeight4FormSensor AND NOT bCountingBeforeSensorsMode);

ftWeight1FormBeforeSensor	(CLK:=bWeight1FormBeforeSensor AND bCountingBeforeSensorsMode AND NOT bWeight1ActuatorSensorUp, Q=>);
ftWeight2FormBeforeSensor	(CLK:=bWeight2FormBeforeSensor AND bCountingBeforeSensorsMode AND NOT bWeight2ActuatorSensorUp, Q=>);
ftWeight3FormBeforeSensor	(CLK:=bWeight3FormBeforeSensor AND bCountingBeforeSensorsMode AND NOT bWeight3ActuatorSensorUp, Q=>);
ftWeight4FormBeforeSensor	(CLK:=bWeight4FormBeforeSensor AND bCountingBeforeSensorsMode AND NOT bWeight4ActuatorSensorUp, Q=>);

//
tonWeightsEmpty			(IN:= iCaseTareWeights = 10 AND NOT bWeight1FormSensor AND NOT bWeight2FormSensor AND NOT bWeight3FormSensor AND NOT bWeight4FormSensor, PT:=T#3S);	
toniCaseTareWeights1	(IN:= iCaseTareWeights = 30, PT:= T#3S);	
toniCaseTareWeights2	(IN:= iCaseTareWeights = 50, PT:= T#3S);	

//=========================================================================================================================================================

//Licznik formatek w górę
tofRunning(IN:= eState = E_Station.eRunning OR eState = E_Station.eStopping OR  eGlobalState=E_PMLState.ePMLState_STOPPING OR eGlobalState=E_PMLState.ePMLState_EXECUTE OR eGlobalState=E_PMLState.ePMLState_STARTING, PT:=T#3S);
//IF eState = E_Station.eRunning OR eState = E_Station.eStopping OR  (eGlobalState=E_PMLState.ePMLState_STOPPING OR eGlobalState=E_PMLState.ePMLState_EXECUTE OR eGlobalState=E_PMLState.ePMLState_STARTING) THEN 
IF tofRunning.Q THEN

	//Liczymy Formatki na Wadze 1 
	IF rtWeight1FormSensor.Q OR ftWeight1FormBeforeSensor.Q THEN
		iFormsCounterWeight1								:= iFormsCounterWeight1 + 1;
	END_IF
	
	//Liczymy Formatki na Wadze 2 
	IF rtWeight2FormSensor.Q OR ftWeight2FormBeforeSensor.Q THEN
		iFormsCounterWeight2								:= iFormsCounterWeight2 + 1;
	END_IF

	//Liczymy Formatki na Wadze 3 
	IF rtWeight3FormSensor.Q OR ftWeight3FormBeforeSensor.Q THEN
		iFormsCounterWeight3								:= iFormsCounterWeight3 + 1;
	END_IF
	
	//Liczymy Formatki na Wadze 4 
	IF rtWeight4FormSensor.Q OR ftWeight4FormBeforeSensor.Q THEN
		iFormsCounterWeight4								:= iFormsCounterWeight4 + 1;
	END_IF

END_IF

//=========================================================================================================================================================
END_ACTION

ACTION ACT_Statistics:

//Statystyka do zliczania czasu cyklu 
rtrigCycleTimerRead(CLK:=bCycleDone);

	IF rtrigCycleTimerRead.Q THEN
		tCycleTime:=tonCycleTimer.ET;
		tt:=tt+1;
	END_IF
	
tonCycleTimer(IN:= eRunningState>E_WeightLiftStationState.eReady , PT:=T#1D);
END_ACTION

ACTION aRepair:
tonRepairOnDelay			(IN:= eState = E_Station.eRunning AND eRunningState = E_WeightLiftStationState.eRepair AND bRepairAllRegistersAreEmpty, PT:= T#2S);

bRepairAllRegistersAreEmpty	:= (NOT arrWeightPackageState[1].bFormPresent AND NOT arrWeightPackageState[2].bFormPresent AND NOT arrWeightPackageState[3].bFormPresent AND NOT arrWeightPackageState[4].bFormPresent);// AND


(** 1 **********************************************************************************************)
tonRepair1(IN:=
									eRunningState = E_WeightLiftStationState.eWeighingCycleON AND
									eState = E_Station.eRunning AND
									bCanReleaseForms AND 
									bConveyorRunning AND 				
									(
									NOT arrWeightPackageState[1].bWeighed OR
									NOT arrWeightPackageState[2].bWeighed OR 
		  							NOT arrWeightPackageState[3].bWeighed OR  
									NOT arrWeightPackageState[4].bWeighed	
									) AND 
									bWeight1FormSensor AND 
									bWeight2FormSensor AND 
									bWeight3FormSensor AND 									
									bWeight4FormSensor 	AND
									NOT tonRepair1.Q							
							, PT:=T#10S);
							
IF 	tonRepair1.Q THEN
	eRunningState		:= E_WeightLiftStationState.eRepair;
	iRepair1 			:= iRepair1	+	1;
END_IF					
(****************************************************************************************************)
(** 2 **********************************************************************************************)
tonRepair2(IN:=
									eRunningState = E_WeightLiftStationState.eStorageOfForms AND
									eState = E_Station.eRunning AND
									bCanReleaseForms AND
									bConveyorRunning AND 
									//(
									//NOT arrWeightPackageState[1].bWeighed OR
									////NOT arrWeightPackageState[2].bWeighed OR 
		  							//NOT arrWeightPackageState[3].bWeighed OR  
									//NOT arrWeightPackageState[4].bWeighed	
									//) AND 
									(
									bWeight1FormSensor OR
									bWeight2FormSensor OR 
									bWeight3FormSensor OR 									
									bWeight4FormSensor 
									) AND
									NOT tonRepair2.Q							
							, PT:=T#10S);
							
IF 	tonRepair2.Q THEN
	eRunningState		:= E_WeightLiftStationState.eRepair;
	iRepair2 			:= iRepair2	+	1;
END_IF					
(****************************************************************************************************)
(** 3 **********************************************************************************************)
tonRepair3(IN:=
									eRunningState = E_WeightLiftStationState.eWeighingCycleON AND
									eState = E_Station.eRunning AND
									bCanReleaseForms AND 
									bConveyorRunning AND 
									(
									NOT arrWeightPackageState[1].bWeighed OR
									NOT arrWeightPackageState[2].bWeighed OR 
		  							NOT arrWeightPackageState[3].bWeighed OR  
									NOT arrWeightPackageState[4].bWeighed	
									) AND 
									NOT bWeight1FormSensor AND 
									NOT bWeight2FormSensor AND 
									NOT bWeight3FormSensor AND 									
									NOT bWeight4FormSensor AND
									NOT tonRepair3.Q							
							, PT:=T#10S);
							
IF 	tonRepair3.Q THEN
	eRunningState		:= E_WeightLiftStationState.eRepair;
	iRepair3 			:= iRepair3	+	1;
END_IF					
(****************************************************************************************************)
(** 4 **********************************************************************************************)
tonRepair4(IN:=
									
									eState = E_Station.eRunning AND
									bCanReleaseForms AND 
									bConveyorRunning AND 
									(
									iFormsCounterWeight1 > 4 OR
									iFormsCounterWeight2 > 4 OR
		  							iFormsCounterWeight3 > 4 OR   
									iFormsCounterWeight4 > 4 
									) AND 
									NOT bWeight1FormSensor AND 
									NOT bWeight2FormSensor AND 
									NOT bWeight3FormSensor AND 									
									NOT bWeight4FormSensor AND
									NOT tonRepair4.Q							
							, PT:=T#10S);
							
IF 	tonRepair4.Q THEN
	eRunningState		:= E_WeightLiftStationState.eRepair;
	iRepair4 			:= iRepair4	+	1;
END_IF					
(****************************************************************************************************)

(** 5 **********************************************************************************************)
tonRepair5(IN:=
									
									eState = E_Station.eRunning AND
									bCanReleaseForms AND
									bConveyorRunning AND 									
									bTwoPhaseMode AND 
									(
									iFormsCounterWeight1 > 2 OR
									iFormsCounterWeight2 > 2 
									) AND 
									//NOT bWeight1FormSensor AND 
									//NOT bWeight2FormSensor AND 

									NOT tonRepair5.Q							
							, PT:=T#8S);
							
IF 	tonRepair5.Q THEN
	eRunningState		:= E_WeightLiftStationState.eRepair;
	iRepair5 			:= iRepair5	+	1;
END_IF					
(****************************************************************************************************)

(** 6 **********************************************************************************************)
tonRepair6(IN:=
									
									(eState = E_Station.eReady OR (eState = E_Station.eRunning AND eRunningState=E_WeightLiftStationState.eStorageOfForms))
									AND
									bCanReleaseForms AND
									bConveyorRunning AND 									
									
									(
									bWeight1Actuator OR
									bWeight2Actuator OR
									bWeight3Actuator OR									
									bWeight4Actuator 								
									) AND 
									NOT tonRepair6.Q							
							, PT:=T#8S);
							
IF 	tonRepair6.Q THEN
	eRunningState			:= E_WeightLiftStationState.eRepair;
	bWeight1Actuator		:= FALSE;
	bWeight2Actuator		:= FALSE;
	bWeight3Actuator		:= FALSE;
	bWeight4Actuator		:= FALSE;	
	iFormsCounterWeight4	:= 0;	
	iFormsCounterWeight3	:= 1;
	iFormsCounterWeight2	:= 2;
	iFormsCounterWeight1	:= 3;	
	iRepair6 				:= iRepair6	+	1;
END_IF					
(****************************************************************************************************)
END_ACTION

ACTION aResetCommands:



bManualWeight1Actuator	:=	FALSE;
bManualWeight2Actuator	:=	FALSE;
bManualWeight3Actuator	:=	FALSE;
bManualWeight4Actuator	:=	FALSE;

bLastStateWeight1Actuator:=	FALSE;
bLastStateWeight2Actuator:=	FALSE;
bLastStateWeight3Actuator:=	FALSE;
bLastStateWeight4Actuator:=	FALSE;

bWeight1Actuator	:=	FALSE;
bWeight2Actuator	:=	FALSE;
bWeight3Actuator	:=	FALSE;
bWeight4Actuator	:=	FALSE;
		

iFormsCounterWeight4	:= 0;	
iFormsCounterWeight3	:= 1;
iFormsCounterWeight2	:= 2;
iFormsCounterWeight1	:= 3;
IF bTwoPhaseMode THEN
	iFormsCounterWeight2	:= 0;
	iFormsCounterWeight1	:= 1;
END_IF


bResetCycleOn			:=	FALSE;	
bWeighingCycleDone		:=	FALSE;
END_ACTION

ACTION aResetCommandsAborting:



bManualWeight1Actuator	:=	FALSE;
bManualWeight2Actuator	:=	FALSE;
bManualWeight3Actuator	:=	FALSE;
bManualWeight4Actuator	:=	FALSE;

bLastStateWeight1Actuator:=	FALSE;
bLastStateWeight2Actuator:=	FALSE;
bLastStateWeight3Actuator:=	FALSE;
bLastStateWeight4Actuator:=	FALSE;

bWeight1Actuator	:=	FALSE;
bWeight2Actuator	:=	FALSE;
bWeight3Actuator	:=	FALSE;
bWeight4Actuator	:=	FALSE;
		

(*iFormsCounterWeight4	:= 0;	
iFormsCounterWeight3	:= 1;
iFormsCounterWeight2	:= 2;
iFormsCounterWeight1	:= 3;
IF bTwoPhaseMode THEN
	iFormsCounterWeight2	:= 0;
	iFormsCounterWeight1	:= 1;
END_IF*)


bResetCycleOn			:=	FALSE;	
bWeighingCycleDone		:=	FALSE;
END_ACTION

ACTION aStationID:
udiStationID	:=	udiStationIndex;
END_ACTION

ACTION ResetAll:
(*****Reset bloczka*****)
IF bEnable THEN
	IF eState <> E_Station.eDisabled AND eState <> E_Station.ePreparingToDisable THEN
		IF bResetCycle THEN
			bResetCycleOn						:= TRUE;
			eState								:= E_Station.ePreparingToReady;
		END_IF
	END_IF
END_IF


IF bResetCycleOn THEN
	
	aResetCommands();
	eRunningState							:= E_WeightLiftStationState.eReady;	
	eState 				 					:= E_Station.eReady;

END_IF
END_ACTION

END_FUNCTION_BLOCK

(* stored: Version 1.1.0.1, ProductVersion 3.1.4026.13, FileIdentifier 6e5447550b69420908d2245a91adb83aa2663c31, FileSignature 6804cf8ea65a47b1bf5a288af89897231f400764c4bff3654cedbf1cb01d3f3fde4fa6e2dffebd6c24878a18848f03a33b3241cf50b4dd0572cd8662a287990095cfe56f753e0930b70556483a6b50749f64d74e973412ae4576a2b81b552d52aab1539edec152804a9f91c4c4fe7a1addefe8d4dc74a9464dbc7bbf304092a465b0f2b00032a94575aee06fdb67e44c9a28386cf3a9b156916771f514e722a99269698751b6568878bcf12320bf7ef9574b5cb2eafb62a37e9e0cd86638ebfab4dc5c9ece3c051b778bbada52602bb21d9f2cf0b046c3f91ddb289cf7364da256cb052932f8ae727ec262c742c4234951bf97a9f2d6f978e731995a6b319028
   POU FB_WeightStation: Id {d0a33ceb-f75d-46b0-a0ca-1b60fad3de25}, SpecialFunc None
   Action ACT_Control: Id {56ebcae9-eff8-4678-9093-23784bb7a1a0}
   Action ACT_ErrorHandling: Id {3b86aa63-9794-4227-978c-cb0f752dfa55}
   Action ACT_Homing: Id {ed2f370f-437b-4851-88fa-9f1cbfb3b23e}
   Action ACT_ManualMovements: Id {2aa08c22-cc09-40c1-8bf7-79e021c798ae}
   Action ACT_Running: Id {312a98c5-9fd2-46c0-bbdd-e5cf8c1c4e70}
   Action ACT_Signals: Id {8f00e1ca-1421-42f5-83e9-cf704a24aaf0}
   Action ACT_Statistics: Id {a6a1e41c-e22e-4888-abf8-da3dd79495c5}
   Action aRepair: Id {2b90b54f-b249-4005-af0c-b96bd82e0684}
   Action aResetCommands: Id {b4b282a3-d87a-417f-ad54-3916058fa3f5}
   Action aResetCommandsAborting: Id {6731ccfc-5885-4da0-aeeb-bfaee88c9365}
   Action aStationID: Id {4b0b40cb-0562-40e0-8ae8-7ca17e4d9db4}
   Action ResetAll: Id {aef51062-c717-4cef-aa55-c0c228733522} *)
